(* Logix 5000 project; controller cal1632 1756-L62 rev 16.20; software revision 16.05; part 15 of 61 *)
(* tags used below, declared in another part *)
   FAULT : BOOL;
   p01_param_temp_limit : REAL;
   p01_sys_scp : SYS_SCP;
   p01r02 : routine;
   p01r09_pb_global_reset : BOOL;
   p12_ai_exhaust_amps : REAL;
   p12_ai_exhaust_hz : REAL;
   p12_ai_exhaust_hz_max : REAL;
   p12_ai_exhaust_rpm : REAL;
   p12_ai_lfl : REAL;
   p12_ai_prs : REAL;
   p12_ai_recirc_amps : REAL;
   p12_ai_recirc_hz : REAL;
   p12_ai_recirc_hz_max : REAL;
   p12_ai_recirc_rpm : REAL;
   p12_ai_tc01 : REAL;
   p12_ai_tc02 : REAL;
   p12_ao_cv : REAL;
   p12_ao_exhaust_selected_speed : REAL;
   p12_ao_recirc_selected_speed : REAL;
   p12_di_burner_auto : BOOL;
   p12_di_burner_safeties_ok : BOOL;
   p12_di_door_open : BOOL;
   p12_di_exh : acs800_di_normal;
   p12_di_exh_fan_mtr_ts : BOOL;
   p12_di_exh_flow_ok : BOOL;
   p12_di_flame_failure : BOOL;
   p12_di_flame_on : BOOL;
   p12_di_fresh_air_clean : BOOL;
   p12_di_high_limit_temp_ok : BOOL;
   p12_di_recirc : acs800_di_normal;
   p12_di_recirc_fan_mtr_ts : BOOL;
   p12_di_recirc_flow_ok : BOOL;
   p12_di_sp0 : BOOL;
   p12_di_sp00 : BOOL;
   p12_di_sp1 : BOOL;
   p12_di_sp2 : BOOL;
   p12_di_sp3 : BOOL;
   p12_di_tc01_bo : BOOL;
   p12_di_tc02_bo : BOOL;
   p12_di_zone_air_clean : BOOL;
   p12_dint_to_hmi : DINT[16];
   p12_do_enable_burner : BOOL;
   p12_do_exh : acs800_do_normal;
   p12_do_recirc : acs800_do_normal;
   p12_do_rst_flame : BOOL;
   p12_exhaust_input_max : REAL;
   p12_exhaust_input_min : REAL;
   p12_exhaust_output_max : REAL;
   p12_exhaust_output_min : REAL;
   p12_hc_input_max : REAL;
   p12_hc_input_min : REAL;
   p12_hc_output_max : REAL;
   p12_hc_output_min : REAL;
   p12_lfl_input_max : REAL;
   p12_lfl_input_min : REAL;
   p12_lfl_output_max : REAL;
   p12_lfl_output_min : REAL;
   p12_param_shutdown_temp : REAL;
   p12_param_tc01z : REAL;
   p12_param_tc02z : REAL;
   p12_param_zone_pressure : REAL;
   p12_prs_input_max : REAL;
   p12_prs_input_min : REAL;
   p12_prs_output_max : REAL;
   p12_prs_output_min : REAL;
   p12_recirc_input_max : REAL;
   p12_recirc_input_min : REAL;
   p12_recirc_output_max : REAL;
   p12_recirc_output_min : REAL;
   p12r01 : routine;
   p12r02 : routine;
   p12r02_fault_exists : BOOL;
   p12r02_not_safe_temp : BOOL;
   p12r02_safe_temp : BOOL;
   p12r02_shutdown_temp : BOOL;
   p12r02_timer_fault : TIMER[4];
   p12r02_timer_safe_temp : TIMER[2];
   p12r02_timer_warning : TIMER[4];
   p12r02_unack_fault : BOOL;
   p12r02_unack_warning : BOOL;
   p12r02_warning_exists : BOOL;
   p12r03 : routine;
   p12r03_hz : SYS_SCP;
   p12r03_timer_fault : TIMER[4];
   p12r03_timer_warning : TIMER[4];
   p12r04 : routine;
   p12r04_timer_fault : TIMER[4];
   p12r04_timer_warning : TIMER[4];
   p12r05 : routine;
   p12r06 : routine;
   p12r07 : routine;
   p12r08 : routine;
   p12r09 : routine;
   p12r10 : routine;
   p12r20 : routine;
   p12r30 : routine;
   p12r30_pb_zone_off : BOOL;
   p12r31 : routine;
   p12r32 : routine;

PROGRAM P12_Zone_2   (* main routine R01_Main *)

ROUTINE R01_Main   (* ladder *)
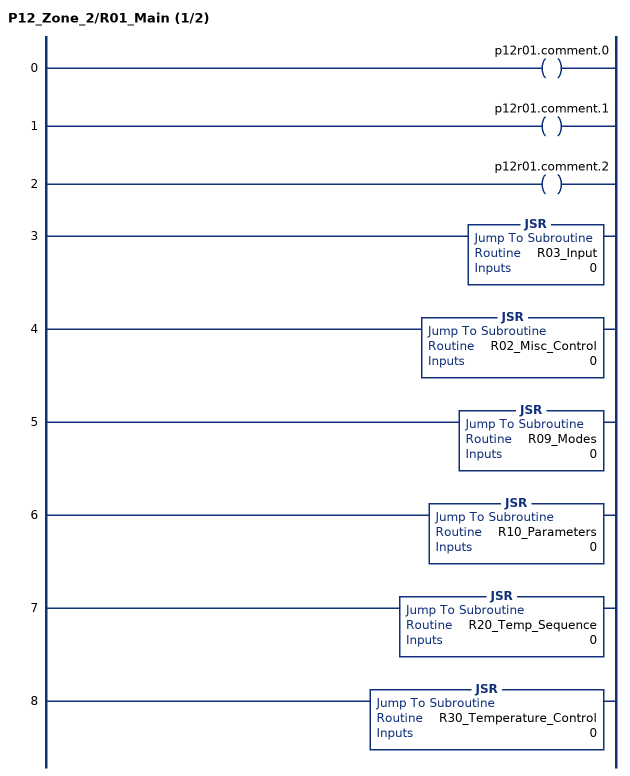
   0: OTE(p12r01.comment.0);
   1: OTE(p12r01.comment.1);
   2: OTE(p12r01.comment.2);
   3: JSR(R03_Input,0);
   4: JSR(R02_Misc_Control,0);
   5: JSR(R09_Modes,0);
   6: JSR(R10_Parameters,0);
   7: JSR(R20_Temp_Sequence,0);
   8: JSR(R30_Temperature_Control,0);
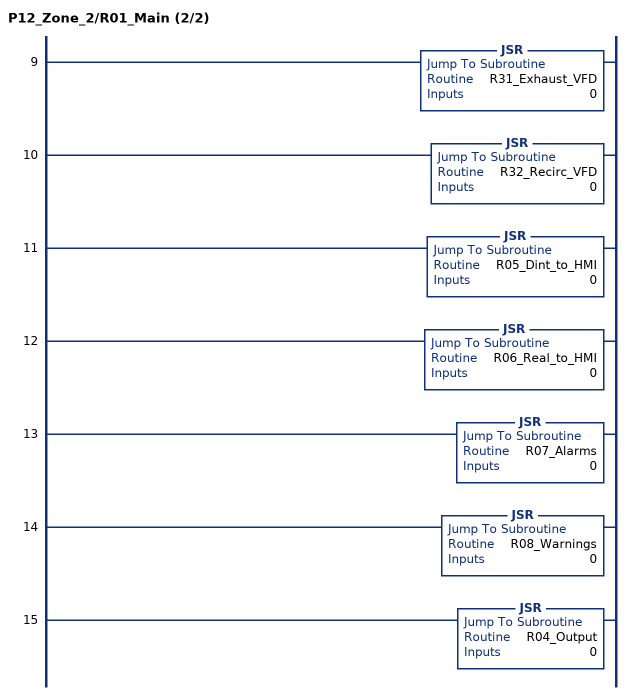
   9: JSR(R31_Exhaust_VFD,0);
   10: JSR(R32_Recirc_VFD,0);
   11: JSR(R05_Dint_to_HMI,0);
   12: JSR(R06_Real_to_HMI,0);
   13: JSR(R07_Alarms,0);
   14: JSR(R08_Warnings,0);
   15: JSR(R04_Output,0);
END_ROUTINE

ROUTINE R02_Misc_Control   (* ladder *)
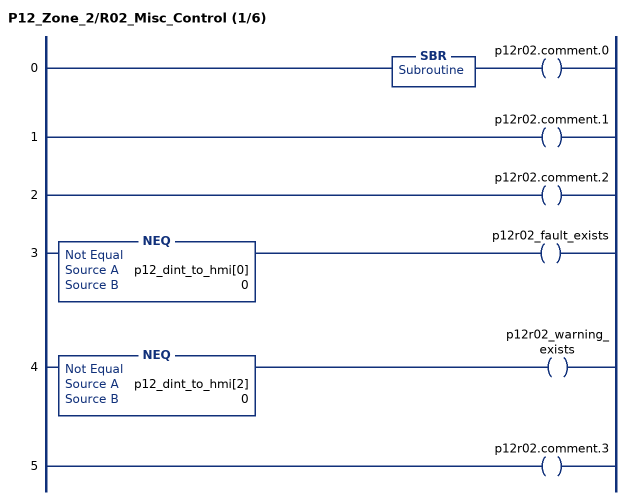
   0: SBR()OTE(p12r02.comment.0);
   1: OTE(p12r02.comment.1);
   2: OTE(p12r02.comment.2);
   3: NEQ(p12_dint_to_hmi[0],0)OTE(p12r02_fault_exists);
   4: NEQ(p12_dint_to_hmi[2],0)OTE(p12r02_warning_exists);
   5: OTE(p12r02.comment.3);
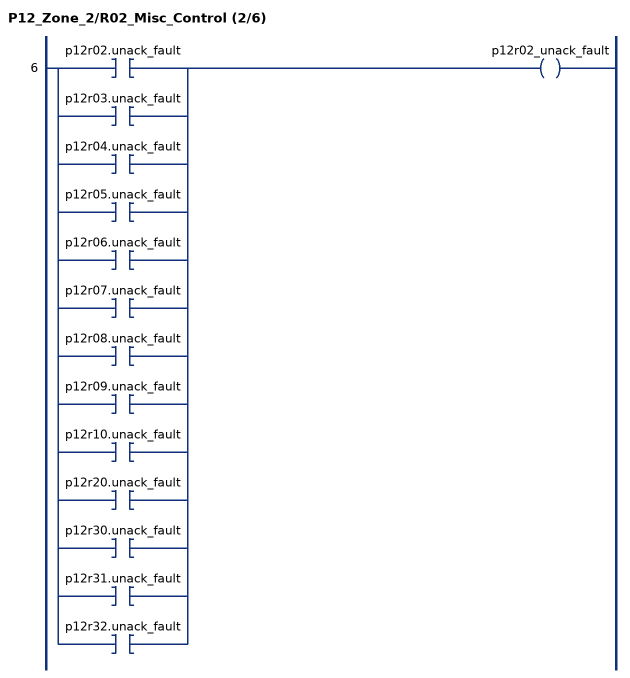
   6: [XIC(p12r02.unack_fault) ,XIC(p12r03.unack_fault) ,XIC(p12r04.unack_fault) ,XIC(p12r05.unack_fault) ,XIC(p12r06.unack_fault) ,XIC(p12r07.unack_fault) ,XIC(p12r08.unack_fault) ,XIC(p12r09.unack_fault) ,XIC(p12r10.unack_fault) ,XIC(p12r20.unack_fault) ,XIC(p12r30.unack_fault) ,XIC(p12r31.unack_fault) ,XIC(p12r32.unack_fault) ]OTE(p12r02_unack_fault);
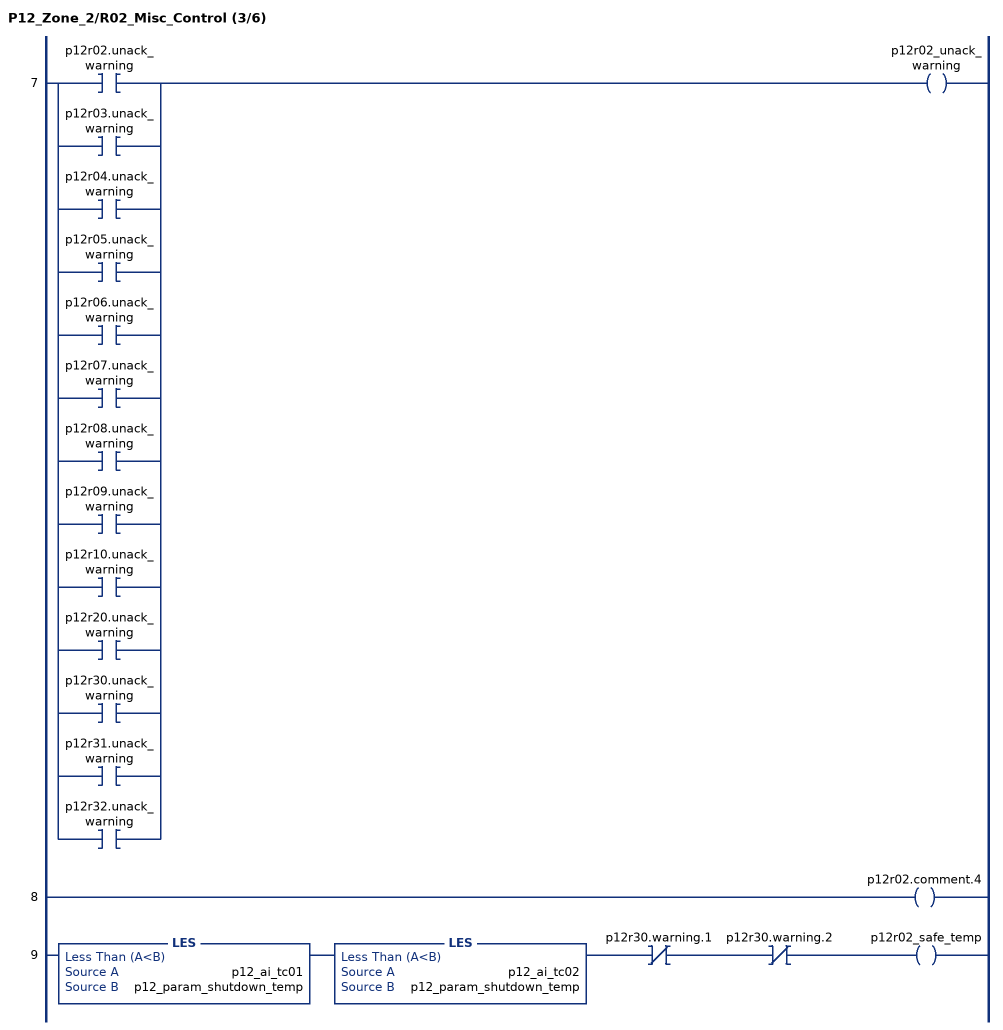
   7: [XIC(p12r02.unack_warning) ,XIC(p12r03.unack_warning) ,XIC(p12r04.unack_warning) ,XIC(p12r05.unack_warning) ,XIC(p12r06.unack_warning) ,XIC(p12r07.unack_warning) ,XIC(p12r08.unack_warning) ,XIC(p12r09.unack_warning) ,XIC(p12r10.unack_warning) ,XIC(p12r20.unack_warning) ,XIC(p12r30.unack_warning) ,XIC(p12r31.unack_warning) ,XIC(p12r32.unack_warning) ]OTE(p12r02_unack_warning);
   8: OTE(p12r02.comment.4);
   9: LES(p12_ai_tc01,p12_param_shutdown_temp)LES(p12_ai_tc02,p12_param_shutdown_temp)XIO(p12r30.warning.1)XIO(p12r30.warning.2)OTE(p12r02_safe_temp);
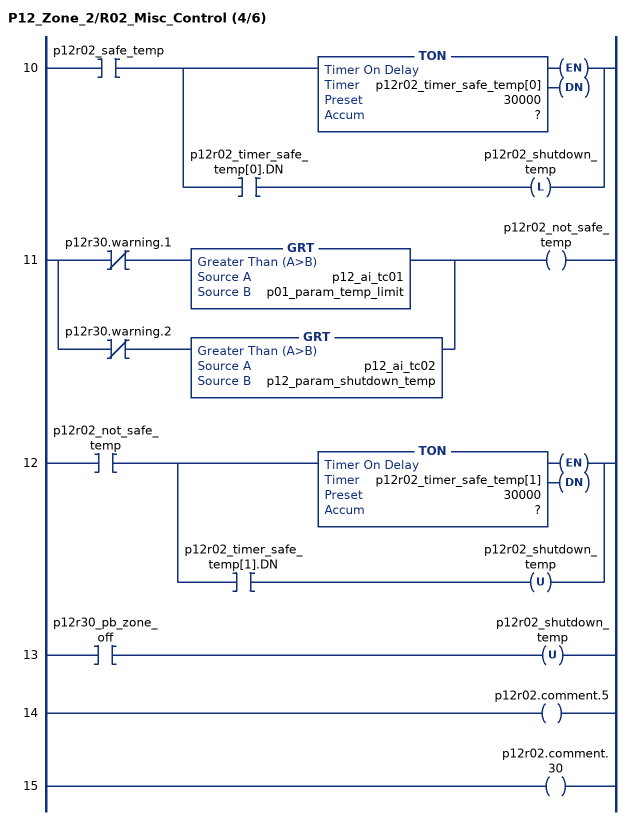
   10: XIC(p12r02_safe_temp)[TON(p12r02_timer_safe_temp[0],?,?) ,XIC(p12r02_timer_safe_temp[0].DN) OTL(p12r02_shutdown_temp) ];
   11: [XIO(p12r30.warning.1) GRT(p12_ai_tc01,p01_param_temp_limit) ,XIO(p12r30.warning.2) GRT(p12_ai_tc02,p12_param_shutdown_temp) ]OTE(p12r02_not_safe_temp);
   12: XIC(p12r02_not_safe_temp)[TON(p12r02_timer_safe_temp[1],?,?) ,XIC(p12r02_timer_safe_temp[1].DN) OTU(p12r02_shutdown_temp) ];
   13: XIC(p12r30_pb_zone_off)OTU(p12r02_shutdown_temp);
   14: OTE(p12r02.comment.5);
   15: OTE(p12r02.comment.30);
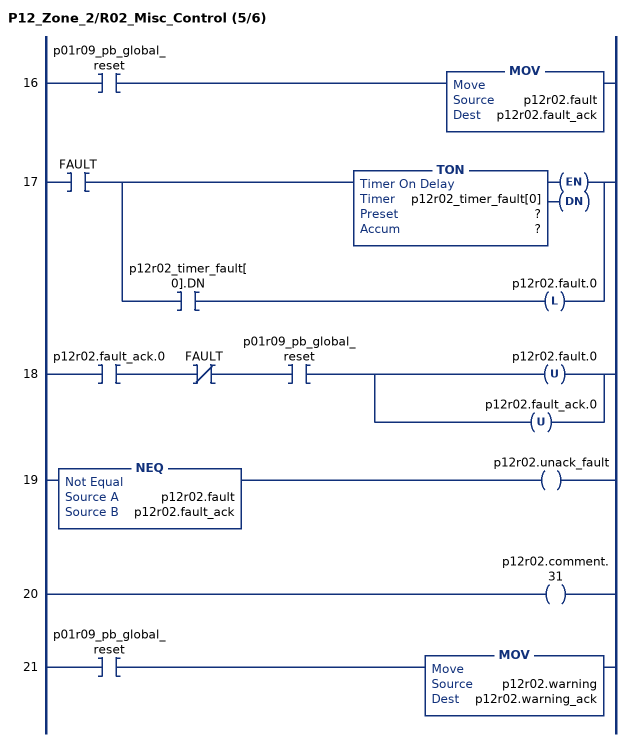
   16: XIC(p01r09_pb_global_reset)MOV(p12r02.fault,p12r02.fault_ack);
   17: XIC(FAULT)[TON(p12r02_timer_fault[0],?,?) ,XIC(p12r02_timer_fault[0].DN) OTL(p12r02.fault.0) ];
   18: XIC(p12r02.fault_ack.0)XIO(FAULT)XIC(p01r09_pb_global_reset)[OTU(p12r02.fault.0) ,OTU(p12r02.fault_ack.0) ];
   19: NEQ(p12r02.fault,p12r02.fault_ack)OTE(p12r02.unack_fault);
   20: OTE(p12r02.comment.31);
   21: XIC(p01r09_pb_global_reset)MOV(p12r02.warning,p12r02.warning_ack);
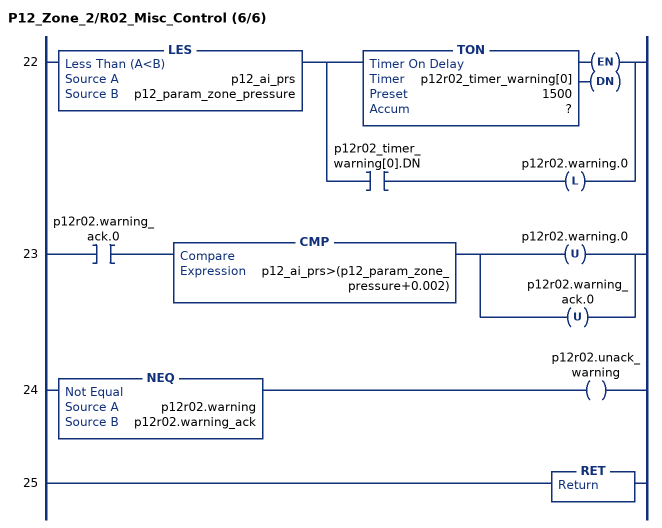
   22: LES(p12_ai_prs,p12_param_zone_pressure)[TON(p12r02_timer_warning[0],?,?) ,XIC(p12r02_timer_warning[0].DN) OTL(p12r02.warning.0) ];
   23: XIC(p12r02.warning_ack.0)CMP(p12_ai_prs>(p12_param_zone_pressure+0.002))[OTU(p12r02.warning.0) ,OTU(p12r02.warning_ack.0) ];
   24: NEQ(p12r02.warning,p12r02.warning_ack)OTE(p12r02.unack_warning);
   25: RET();
END_ROUTINE

ROUTINE R03_Input   (* ladder *)
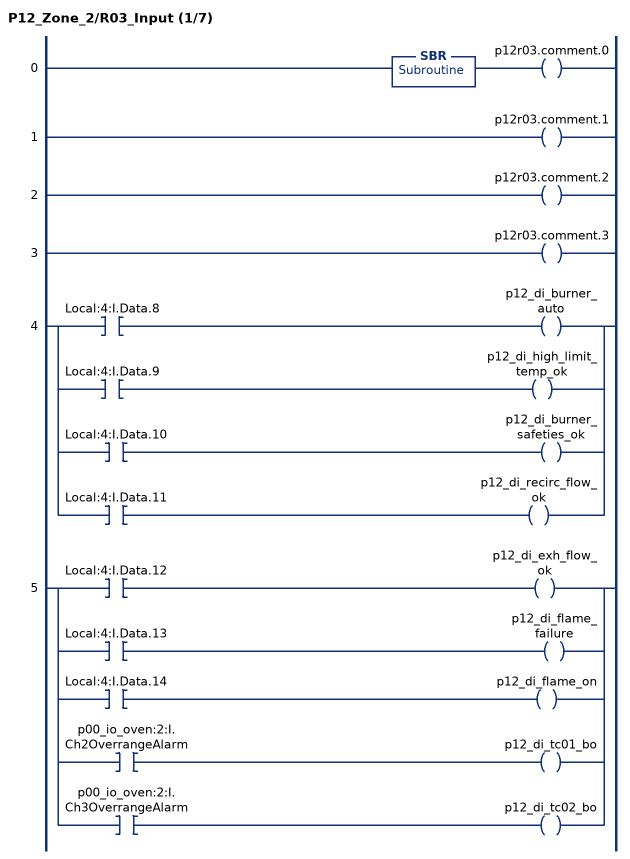
   0: SBR()OTE(p12r03.comment.0);
   1: OTE(p12r03.comment.1);
   2: OTE(p12r03.comment.2);
   3: OTE(p12r03.comment.3);
   4: [XIC(Local:4:I.Data.8) OTE(p12_di_burner_auto) ,XIC(Local:4:I.Data.9) OTE(p12_di_high_limit_temp_ok) ,XIC(Local:4:I.Data.10) OTE(p12_di_burner_safeties_ok) ,XIC(Local:4:I.Data.11) OTE(p12_di_recirc_flow_ok) ];
   5: [XIC(Local:4:I.Data.12) OTE(p12_di_exh_flow_ok) ,XIC(Local:4:I.Data.13) OTE(p12_di_flame_failure) ,XIC(Local:4:I.Data.14) OTE(p12_di_flame_on) ,XIC(p00_io_oven:2:I.Ch2OverrangeAlarm) OTE(p12_di_tc01_bo) ,XIC(p00_io_oven:2:I.Ch3OverrangeAlarm) OTE(p12_di_tc02_bo) ];
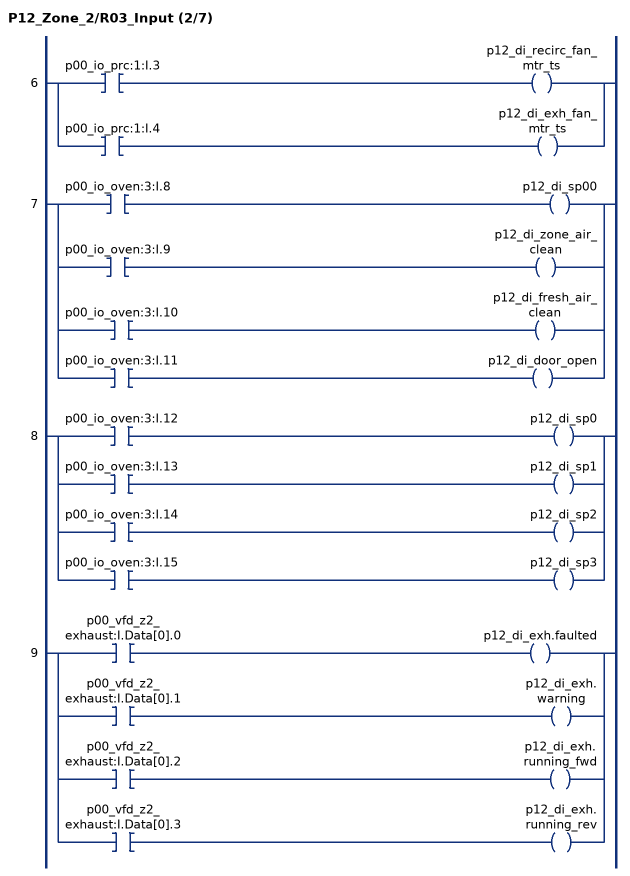
   6: [XIC(p00_io_prc:1:I.3) OTE(p12_di_recirc_fan_mtr_ts) ,XIC(p00_io_prc:1:I.4) OTE(p12_di_exh_fan_mtr_ts) ];
   7: [XIC(p00_io_oven:3:I.8) OTE(p12_di_sp00) ,XIC(p00_io_oven:3:I.9) OTE(p12_di_zone_air_clean) ,XIC(p00_io_oven:3:I.10) OTE(p12_di_fresh_air_clean) ,XIC(p00_io_oven:3:I.11) OTE(p12_di_door_open) ];
   8: [XIC(p00_io_oven:3:I.12) OTE(p12_di_sp0) ,XIC(p00_io_oven:3:I.13) OTE(p12_di_sp1) ,XIC(p00_io_oven:3:I.14) OTE(p12_di_sp2) ,XIC(p00_io_oven:3:I.15) OTE(p12_di_sp3) ];
   9: [XIC(p00_vfd_z2_exhaust:I.Data[0].0) OTE(p12_di_exh.faulted) ,XIC(p00_vfd_z2_exhaust:I.Data[0].1) OTE(p12_di_exh.warning) ,XIC(p00_vfd_z2_exhaust:I.Data[0].2) OTE(p12_di_exh.running_fwd) ,XIC(p00_vfd_z2_exhaust:I.Data[0].3) OTE(p12_di_exh.running_rev) ];
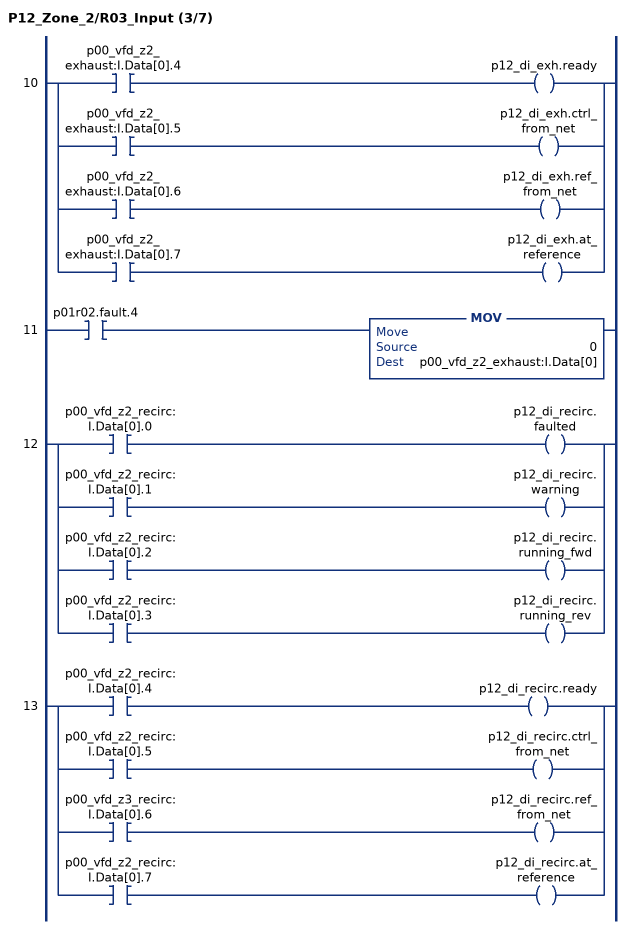
   10: [XIC(p00_vfd_z2_exhaust:I.Data[0].4) OTE(p12_di_exh.ready) ,XIC(p00_vfd_z2_exhaust:I.Data[0].5) OTE(p12_di_exh.ctrl_from_net) ,XIC(p00_vfd_z2_exhaust:I.Data[0].6) OTE(p12_di_exh.ref_from_net) ,XIC(p00_vfd_z2_exhaust:I.Data[0].7) OTE(p12_di_exh.at_reference) ];
   11: XIC(p01r02.fault.4)MOV(0,p00_vfd_z2_exhaust:I.Data[0]);
   12: [XIC(p00_vfd_z2_recirc:I.Data[0].0) OTE(p12_di_recirc.faulted) ,XIC(p00_vfd_z2_recirc:I.Data[0].1) OTE(p12_di_recirc.warning) ,XIC(p00_vfd_z2_recirc:I.Data[0].2) OTE(p12_di_recirc.running_fwd) ,XIC(p00_vfd_z2_recirc:I.Data[0].3) OTE(p12_di_recirc.running_rev) ];
   13: [XIC(p00_vfd_z2_recirc:I.Data[0].4) OTE(p12_di_recirc.ready) ,XIC(p00_vfd_z2_recirc:I.Data[0].5) OTE(p12_di_recirc.ctrl_from_net) ,XIC(p00_vfd_z3_recirc:I.Data[0].6) OTE(p12_di_recirc.ref_from_net) ,XIC(p00_vfd_z2_recirc:I.Data[0].7) OTE(p12_di_recirc.at_reference) ];
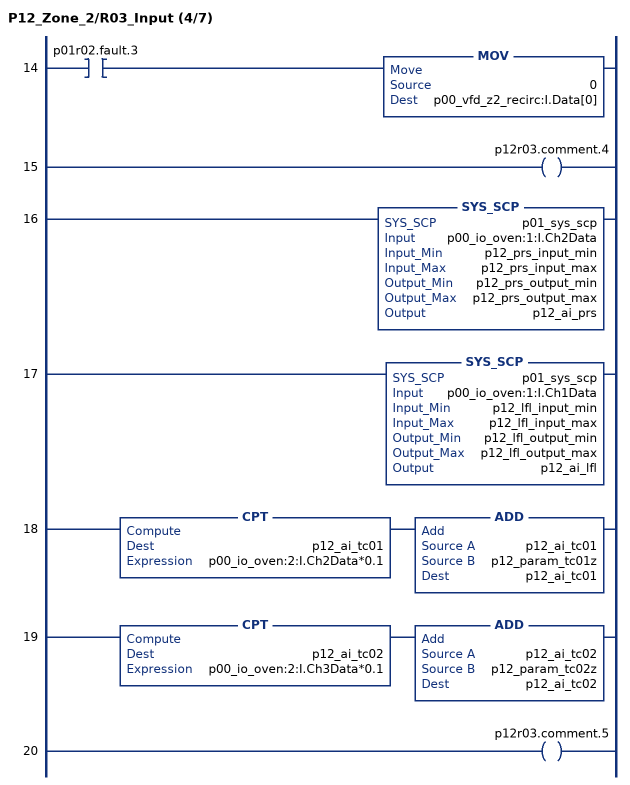
   14: XIC(p01r02.fault.3)MOV(0,p00_vfd_z2_recirc:I.Data[0]);
   15: OTE(p12r03.comment.4);
   16: SYS_SCP(p01_sys_scp,p00_io_oven:1:I.Ch2Data,p12_prs_input_min,p12_prs_input_max,p12_prs_output_min,p12_prs_output_max,p12_ai_prs);
   17: SYS_SCP(p01_sys_scp,p00_io_oven:1:I.Ch1Data,p12_lfl_input_min,p12_lfl_input_max,p12_lfl_output_min,p12_lfl_output_max,p12_ai_lfl);
   18: CPT(p12_ai_tc01,p00_io_oven:2:I.Ch2Data*0.1)ADD(p12_ai_tc01,p12_param_tc01z,p12_ai_tc01);
   19: CPT(p12_ai_tc02,p00_io_oven:2:I.Ch3Data*0.1)ADD(p12_ai_tc02,p12_param_tc02z,p12_ai_tc02);
   20: OTE(p12r03.comment.5);
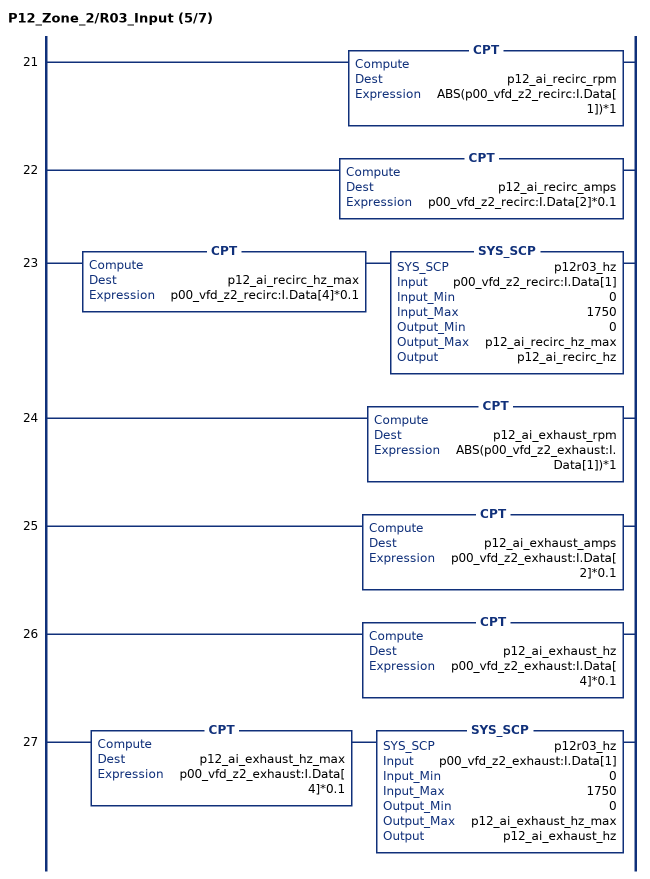
   21: CPT(p12_ai_recirc_rpm,ABS(p00_vfd_z2_recirc:I.Data[1])*1);
   22: CPT(p12_ai_recirc_amps,p00_vfd_z2_recirc:I.Data[2]*0.1);
   23: CPT(p12_ai_recirc_hz_max,p00_vfd_z2_recirc:I.Data[4]*0.1)SYS_SCP(p12r03_hz,p00_vfd_z2_recirc:I.Data[1],0,1750,0,p12_ai_recirc_hz_max,p12_ai_recirc_hz);
   24: CPT(p12_ai_exhaust_rpm,ABS(p00_vfd_z2_exhaust:I.Data[1])*1);
   25: CPT(p12_ai_exhaust_amps,p00_vfd_z2_exhaust:I.Data[2]*0.1);
   26: CPT(p12_ai_exhaust_hz,p00_vfd_z2_exhaust:I.Data[4]*0.1);
   27: CPT(p12_ai_exhaust_hz_max,p00_vfd_z2_exhaust:I.Data[4]*0.1)SYS_SCP(p12r03_hz,p00_vfd_z2_exhaust:I.Data[1],0,1750,0,p12_ai_exhaust_hz_max,p12_ai_exhaust_hz);
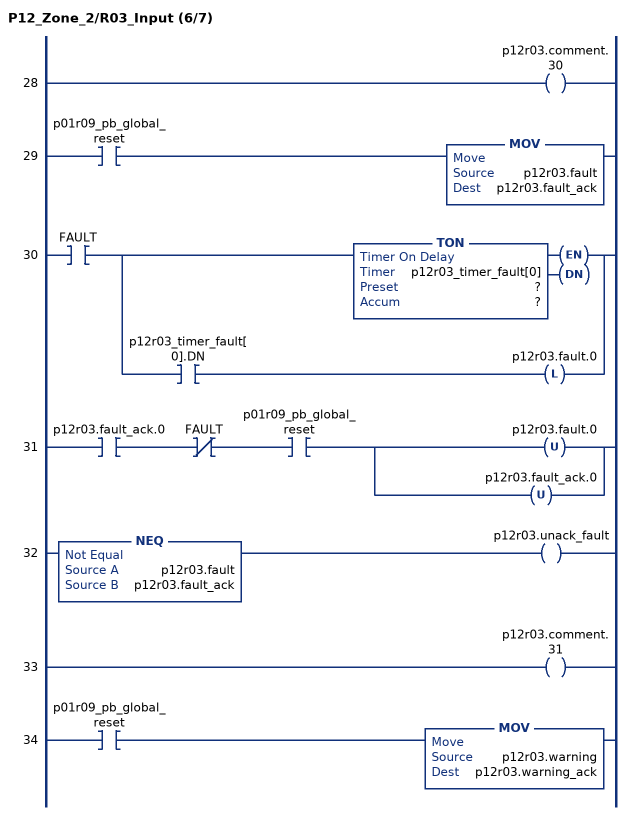
   28: OTE(p12r03.comment.30);
   29: XIC(p01r09_pb_global_reset)MOV(p12r03.fault,p12r03.fault_ack);
   30: XIC(FAULT)[TON(p12r03_timer_fault[0],?,?) ,XIC(p12r03_timer_fault[0].DN) OTL(p12r03.fault.0) ];
   31: XIC(p12r03.fault_ack.0)XIO(FAULT)XIC(p01r09_pb_global_reset)[OTU(p12r03.fault.0) ,OTU(p12r03.fault_ack.0) ];
   32: NEQ(p12r03.fault,p12r03.fault_ack)OTE(p12r03.unack_fault);
   33: OTE(p12r03.comment.31);
   34: XIC(p01r09_pb_global_reset)MOV(p12r03.warning,p12r03.warning_ack);
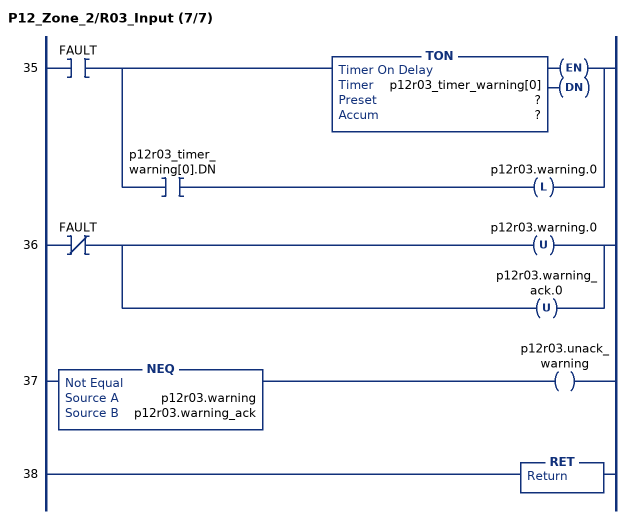
   35: XIC(FAULT)[TON(p12r03_timer_warning[0],?,?) ,XIC(p12r03_timer_warning[0].DN) OTL(p12r03.warning.0) ];
   36: XIO(FAULT)[OTU(p12r03.warning.0) ,OTU(p12r03.warning_ack.0) ];
   37: NEQ(p12r03.warning,p12r03.warning_ack)OTE(p12r03.unack_warning);
   38: RET();
END_ROUTINE

ROUTINE R04_Output   (* ladder *)
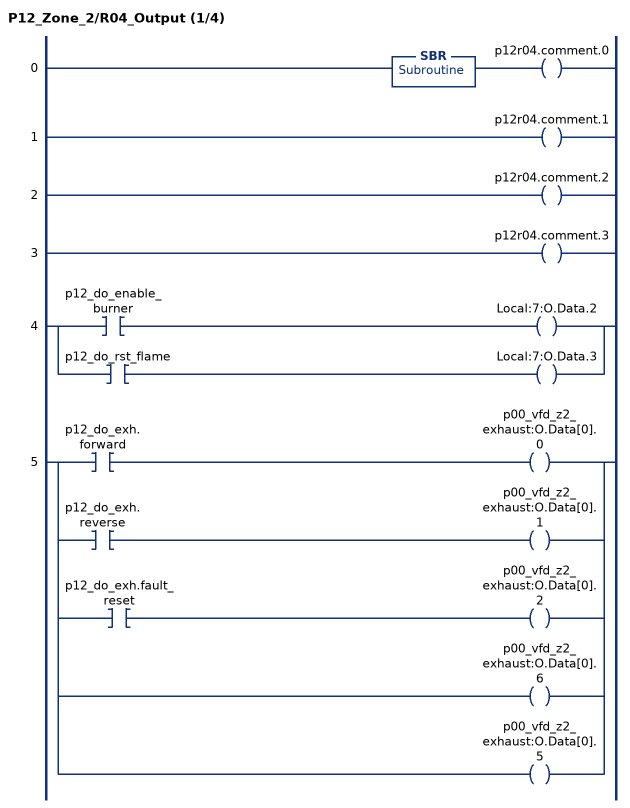
   0: SBR()OTE(p12r04.comment.0);
   1: OTE(p12r04.comment.1);
   2: OTE(p12r04.comment.2);
   3: OTE(p12r04.comment.3);
   4: [XIC(p12_do_enable_burner) OTE(Local:7:O.Data.2) ,XIC(p12_do_rst_flame) OTE(Local:7:O.Data.3) ];
   5: [XIC(p12_do_exh.forward) OTE(p00_vfd_z2_exhaust:O.Data[0].0) ,XIC(p12_do_exh.reverse) OTE(p00_vfd_z2_exhaust:O.Data[0].1) ,XIC(p12_do_exh.fault_reset) OTE(p00_vfd_z2_exhaust:O.Data[0].2) ,OTE(p00_vfd_z2_exhaust:O.Data[0].6) ,OTE(p00_vfd_z2_exhaust:O.Data[0].5) ];
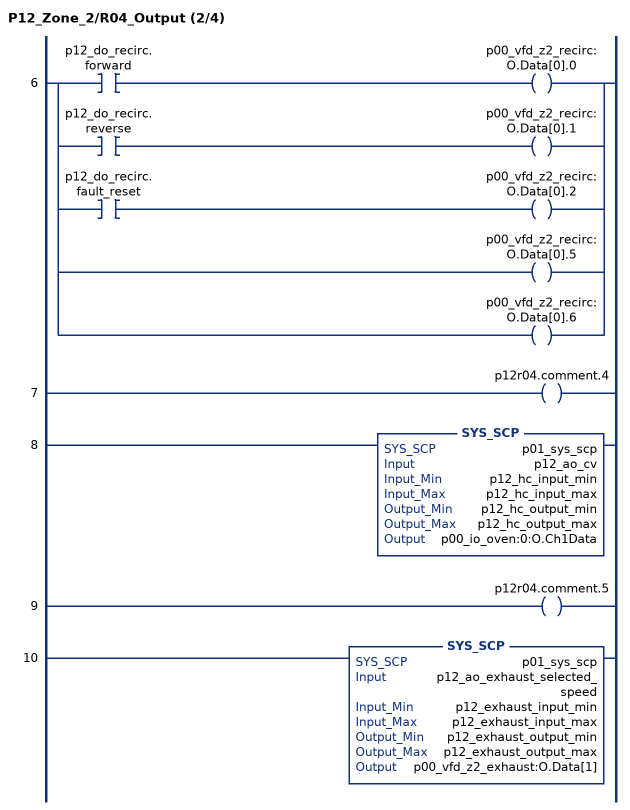
   6: [XIC(p12_do_recirc.forward) OTE(p00_vfd_z2_recirc:O.Data[0].0) ,XIC(p12_do_recirc.reverse) OTE(p00_vfd_z2_recirc:O.Data[0].1) ,XIC(p12_do_recirc.fault_reset) OTE(p00_vfd_z2_recirc:O.Data[0].2) ,OTE(p00_vfd_z2_recirc:O.Data[0].5) ,OTE(p00_vfd_z2_recirc:O.Data[0].6) ];
   7: OTE(p12r04.comment.4);
   8: SYS_SCP(p01_sys_scp,p12_ao_cv,p12_hc_input_min,p12_hc_input_max,p12_hc_output_min,p12_hc_output_max,p00_io_oven:0:O.Ch1Data);
   9: OTE(p12r04.comment.5);
   10: SYS_SCP(p01_sys_scp,p12_ao_exhaust_selected_speed,p12_exhaust_input_min,p12_exhaust_input_max,p12_exhaust_output_min,p12_exhaust_output_max,p00_vfd_z2_exhaust:O.Data[1]);
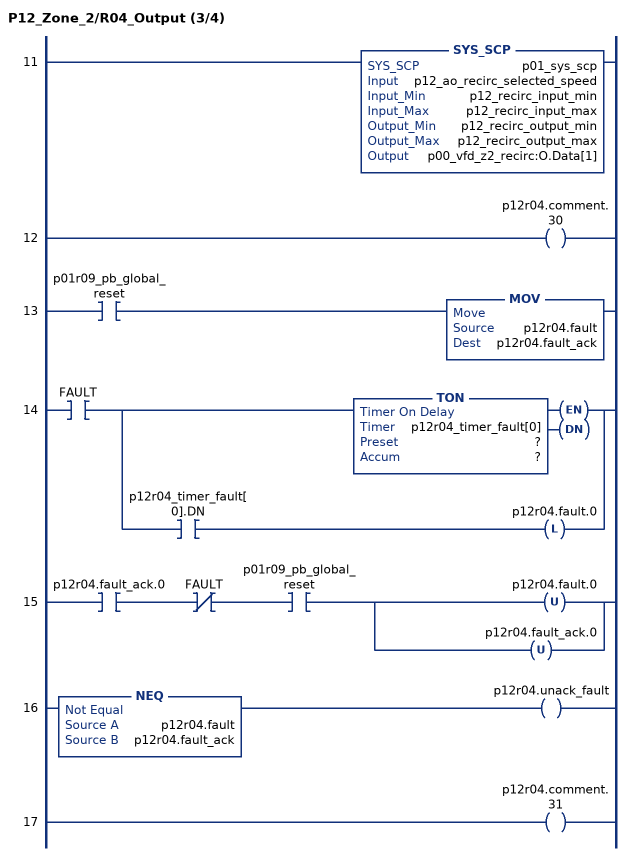
   11: SYS_SCP(p01_sys_scp,p12_ao_recirc_selected_speed,p12_recirc_input_min,p12_recirc_input_max,p12_recirc_output_min,p12_recirc_output_max,p00_vfd_z2_recirc:O.Data[1]);
   12: OTE(p12r04.comment.30);
   13: XIC(p01r09_pb_global_reset)MOV(p12r04.fault,p12r04.fault_ack);
   14: XIC(FAULT)[TON(p12r04_timer_fault[0],?,?) ,XIC(p12r04_timer_fault[0].DN) OTL(p12r04.fault.0) ];
   15: XIC(p12r04.fault_ack.0)XIO(FAULT)XIC(p01r09_pb_global_reset)[OTU(p12r04.fault.0) ,OTU(p12r04.fault_ack.0) ];
   16: NEQ(p12r04.fault,p12r04.fault_ack)OTE(p12r04.unack_fault);
   17: OTE(p12r04.comment.31);
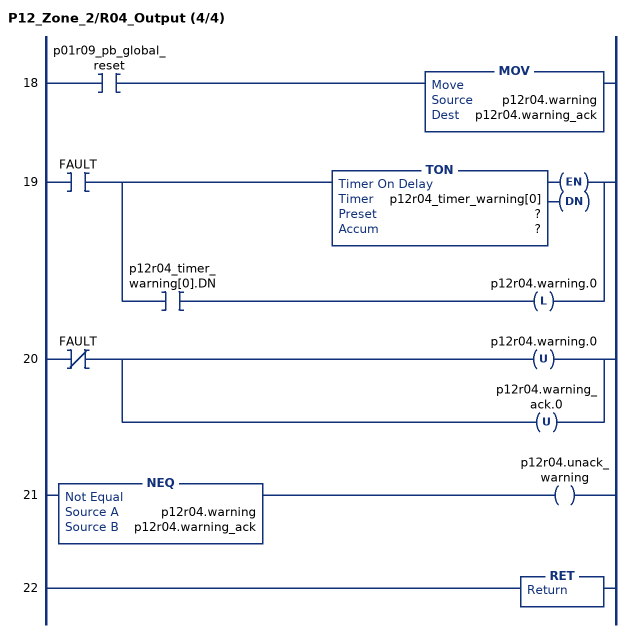
   18: XIC(p01r09_pb_global_reset)MOV(p12r04.warning,p12r04.warning_ack);
   19: XIC(FAULT)[TON(p12r04_timer_warning[0],?,?) ,XIC(p12r04_timer_warning[0].DN) OTL(p12r04.warning.0) ];
   20: XIO(FAULT)[OTU(p12r04.warning.0) ,OTU(p12r04.warning_ack.0) ];
   21: NEQ(p12r04.warning,p12r04.warning_ack)OTE(p12r04.unack_warning);
   22: RET();
END_ROUTINE
